(* IEC 61131-3 sources: AXOpen/src/integrations/app/src/Examples/AXOpen.Cognex.Vision, 2 files *)

(* ---- AxoCognexVisionDatamanExample.st ---- *)
USING AXOpen.Core;
USING AXOpen.Components.Cognex.Vision.v_6_0_0_0;

NAMESPACE AxoCognexVisionDatamanExamples

    {S7.extern=ReadWrite}
    CLASS AxoCognexVisionDatamanExampleContext EXTENDS AXOpen.Core.AxoContext
        VAR PUBLIC
            {#ix-set:AttributeName = "10A1"}
            MyDataman1 : AXOpen.Components.Cognex.Vision.v_6_0_0_0.AxoDataman;
            {#ix-set:AttributeName = "reader_st2"}
            MyDataman2 : AXOpen.Components.Cognex.Vision.v_6_0_0_0.AxoDataman;
            {#ix-set:AttributeName = "<#Activate manual control#>"}
            ActivateManualControl : BOOL;
            myString : STRING;
            _rootObject :   AxoObject;
        END_VAR

        METHOD PROTECTED OVERRIDE Main
            // Example of the activation of the manual control.
            IF ActivateManualControl THEN
                MyDataman1.ActivateManualControl();
                MyDataman2.ActivateManualControl();
            END_IF;
            // Calling the main method `Run` with respective input and output variables.
            THIS.InitializeRootObject(_rootObject);
            //<HWIO_Assignement>
            MyDataman1.Run( parent                     :=  _rootObject,
                            ResultDataSize             :=  AXOpen.Components.Cognex.Vision.v_6_0_0_0.eAxoDataman_ResultDataSize#RESULT_DATA_128B,
                            UserDataSize               :=  AXOpen.Components.Cognex.Vision.v_6_0_0_0.eAxoDataman_UserDataSize#USER_DATA_128B,
                            hwID                       :=  HwIdentifiers#_10a1,
                            hwIdAcquisitionControl     :=  HwIdentifiers#_10a1_Acquisition_Control_1,
                            hwIdAcquisitionStatus      :=  HwIdentifiers#_10a1_Acquisition_Status_1,
                            hwIdResultsControl         :=  HwIdentifiers#_10a1_Results_Control_1,
                            hwIdResultsStatus          :=  HwIdentifiers#_10a1_Results_Status_1,
                            hwIdSoftEventControl       :=  HwIdentifiers#_10a1_Soft_Event_Control_1,
                            hwIdResultData             :=  HwIdentifiers#_10a1_Result_Data_128_bytes_1,
                            hwIdUserData               :=  HwIdentifiers#_10a1_User_Data_128_bytes_1);
            //</HWIO_Assignement>
            MyDataman2.Run( parent                     :=  _rootObject,
                            ResultDataSize             :=  AXOpen.Components.Cognex.Vision.v_6_0_0_0.eAxoDataman_ResultDataSize#RESULT_DATA_64B,
                            UserDataSize               :=  AXOpen.Components.Cognex.Vision.v_6_0_0_0.eAxoDataman_UserDataSize#USER_DATA_64B,
                            hwID                       :=  HwIdentifiers#reader_st2,
                            hwIdAcquisitionControl     :=  HwIdentifiers#reader_st2_Acquisition_Control_1,
                            hwIdAcquisitionStatus      :=  HwIdentifiers#reader_st2_Acquisition_Status_1,
                            hwIdResultsControl         :=  HwIdentifiers#reader_st2_Results_Control_1,
                            hwIdResultsStatus          :=  HwIdentifiers#reader_st2_Results_Status_1,
                            hwIdSoftEventControl       :=  HwIdentifiers#reader_st2_Soft_Event_Control_1,
                            hwIdResultData             :=  HwIdentifiers#reader_st2_Result_Data_64_bytes_1,
                            hwIdUserData               :=  HwIdentifiers#reader_st2_User_Data_64_bytes_1);

        END_METHOD

        METHOD DocuExample
                //<Read>
                IF MyDataman1.Read().IsDone() THEN
                    //Process the result data
                    // myString := MyDataman1.ResultData.Data;
                    ;
                END_IF;
                //</Read>

                //<ClearResultData>
                IF MyDataman1.ClearResultData().IsDone() THEN
                    //Data inside MyDataman1.Results.Data is cleared
                    ;
                END_IF;
                //</ClearResultData>
        END_METHOD

    END_CLASS
END_NAMESPACE

(* ---- AxoCognexVisionInsightExample.st ---- *)
USING AXOpen.Core;
USING AXOpen.Components.Cognex.Vision.v_6_0_0_0;

NAMESPACE AxoCognexVisionInsightExamples

    {S7.extern=ReadWrite}
    CLASS AxoCognexVisionInsightExampleContext EXTENDS AXOpen.Core.AxoContext
        VAR PUBLIC
            {#ix-set:AttributeName = "someInsight"}
            MyInsight : AXOpen.Components.Cognex.Vision.v_6_0_0_0.AxoInsight;
            {#ix-set:AttributeName = "<#Activate manual control#>"}
            ActivateManualControl : BOOL;
            _rootObject :   AxoObject;
        END_VAR

        METHOD PROTECTED OVERRIDE Main
            // Example of the activation of the manual control.
            IF ActivateManualControl THEN
                MyInsight.ActivateManualControl();
            END_IF;
            // Calling the main method `Run` with respective input and output variables.
            _rootObject.InitializeWithContext(THIS);
            //<HWIO_Assignement>
            MyInsight.Run(  parent                  :=  _rootObject,
                            ResultDataSize          :=  AXOpen.Components.Cognex.Vision.v_6_0_0_0.eAxoInsight_ResultDataSize#RESULT_DATA_64B,
                            UserDataSize            :=  AXOpen.Components.Cognex.Vision.v_6_0_0_0.eAxoInsight_UserDataSize#USER_DATA_64B,
                            hwID                    :=  HwIdentifiers#_7600,
                            hwIdAcquisitionControl  :=  HwIdentifiers#_7600_Acquisition_Control_1,
                            hwIdAcquisitionStatus   :=  HwIdentifiers#_7600_Acquisition_Status_1,
                            hwIdInspectionControl   :=  HwIdentifiers#_7600_Inspection_Control_1,
                            hwIdInspectionStatus    :=  HwIdentifiers#_7600_Inspection_Status_1,
                            hwIdCommandControl      :=  HwIdentifiers#_7600_Command_Control_1,
                            hwIdSoftEventControl    :=  HwIdentifiers#_7600_SoftEvent_Control_1,
                            hwIdResultData          :=  HwIdentifiers#_7600_Results_64_bytes_1,
                            hwIdUserData            :=  HwIdentifiers#_7600_User_Data_64_bytes_1);
            //</HWIO_Assignement>
        END_METHOD

        METHOD DocuExample
            VAR
                myData : ARRAY[0..249] OF BYTE;
            END_VAR

                //<ClearInspectionResults>
                IF MyInsight.ClearInspectionResults().IsDone() THEN
                    //Data inside MyInsight.InspectionResults.Data is cleared
                    ;
                END_IF;
                //</ClearInspectionResults>

                //<Trigger>
                IF MyInsight.Trigger().IsDone() THEN
                    //Process the result data
                    myData := MyInsight.InspectionResults.Data;
                END_IF;
                //</Trigger>

                //<ChangeJobByNumber>
                IF MyInsight.ChangeJob(UINT#5).IsDone() THEN
                    ;
                END_IF;
                //</ChangeJobByNumber>

                //<ChangeJobByName>
                IF MyInsight.ChangeJob('MyJobName.job').IsDone() THEN
                    ;
                END_IF;
                //</ChangeJobByName>

                //<SoftEvent>
                IF MyInsight.SoftEvent(UINT#5).IsDone() THEN
                    ;
                END_IF;
                //</SoftEvent>

        END_METHOD

    END_CLASS
END_NAMESPACE
